% RSLogix 500 project P2.RSS, saved by version 8.30.00.16 %
PROJECT "UNTITLED"    % processor: Bul.1763 MicroLogix 1100 Series B %

PROGRAM FILES
  LAD 2 "MAIN"  3 rungs
  LAD 3 "IO"  9 rungs
  LAD 4 "CONTROLS"  9 rungs

DATA FILES
  O0 OUTPUT  4 elements
  I1 INPUT  6 elements
  S2 STATUS  66 elements
  B3 BINARY  1 elements
  T4 TIMER  2 elements
  C5 COUNTER  1 elements
  R6 CONTROL  1 elements
  N7 INTEGER  1 elements
  F8 FLOAT  1 elements

LADDER 2 "MAIN"
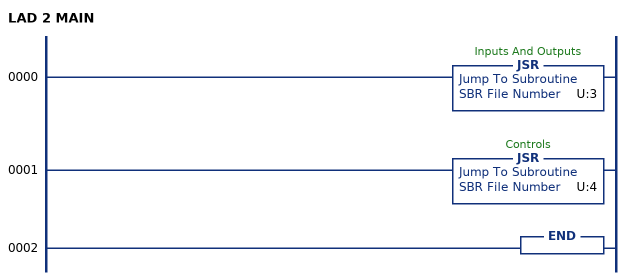
% Rung: 0 %
SOR JSR U:3 EOR
%   U:3  "Inputs And Outputs" %
% Rung: 1 %
SOR JSR U:4 EOR
%   U:4  "Controls" %
% Rung: 2 %
SOR END EOR

LADDER 3 "IO"
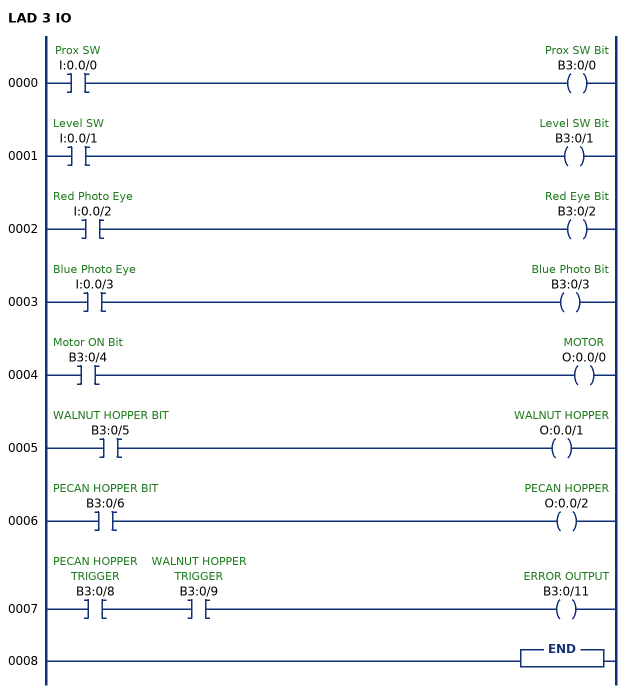
% Rung: 0 %
SOR XIC I:0.0/0 OTE B3:0/0 EOR
%   I:0.0/0  "Prox SW" %
%   B3:0/0  "Prox SW Bit" %
% Rung: 1 %
SOR XIC I:0.0/1 OTE B3:0/1 EOR
%   I:0.0/1  "Level SW" %
%   B3:0/1  "Level SW Bit" %
% Rung: 2 %
SOR XIC I:0.0/2 OTE B3:0/2 EOR
%   I:0.0/2  "Red Photo Eye" %
%   B3:0/2  "Red Eye Bit" %
% Rung: 3 %
SOR XIC I:0.0/3 OTE B3:0/3 EOR
%   I:0.0/3  "Blue Photo Eye" %
%   B3:0/3  "Blue Photo Bit" %
% Rung: 4 %
SOR XIC B3:0/4 OTE O:0.0/0 EOR
%   B3:0/4  "Motor ON Bit" %
%   O:0.0/0  "MOTOR" %
% Rung: 5 %
SOR XIC B3:0/5 OTE O:0.0/1 EOR
%   B3:0/5  "WALNUT HOPPER BIT" %
%   O:0.0/1  "WALNUT HOPPER" %
% Rung: 6 %
SOR XIC B3:0/6 OTE O:0.0/2 EOR
%   B3:0/6  "PECAN HOPPER BIT" %
%   O:0.0/2  "PECAN HOPPER" %
% Rung: 7 %
SOR XIC B3:0/8 XIC B3:0/9 OTE B3:0/11 EOR
%   B3:0/8  "PECAN HOPPER TRIGGER" %
%   B3:0/9  "WALNUT HOPPER TRIGGER" %
%   B3:0/11  "ERROR OUTPUT" %
% Rung: 8 %
SOR END EOR

LADDER 4 "CONTROLS"
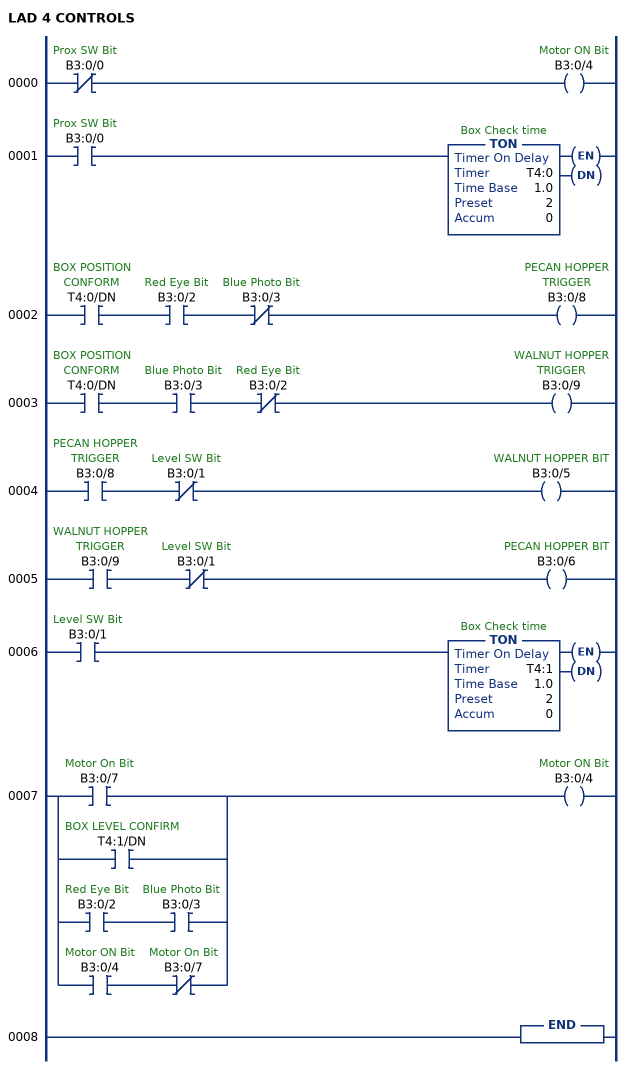
% Rung: 0 %
SOR XIO B3:0/0 OTE B3:0/4 EOR
%   B3:0/0  "Prox SW Bit" %
%   B3:0/4  "Motor ON Bit" %
% Rung: 1 %
SOR XIC B3:0/0 TON T4:0 1.0 2 0 EOR
%   B3:0/0  "Prox SW Bit" %
%   T4:0  "Box Check time" %
% Rung: 2 %
SOR XIC T4:0/DN XIC B3:0/2 XIO B3:0/3 OTE B3:0/8 EOR
%   T4:0/DN  "BOX POSITION CONFORM" %
%   B3:0/2  "Red Eye Bit" %
%   B3:0/3  "Blue Photo Bit" %
%   B3:0/8  "PECAN HOPPER TRIGGER" %
% Rung: 3 %
SOR XIC T4:0/DN XIC B3:0/3 XIO B3:0/2 OTE B3:0/9 EOR
%   T4:0/DN  "BOX POSITION CONFORM" %
%   B3:0/3  "Blue Photo Bit" %
%   B3:0/2  "Red Eye Bit" %
%   B3:0/9  "WALNUT HOPPER TRIGGER" %
% Rung: 4 %
SOR XIC B3:0/8 XIO B3:0/1 OTE B3:0/5 EOR
%   B3:0/8  "PECAN HOPPER TRIGGER" %
%   B3:0/1  "Level SW Bit" %
%   B3:0/5  "WALNUT HOPPER BIT" %
% Rung: 5 %
SOR XIC B3:0/9 XIO B3:0/1 OTE B3:0/6 EOR
%   B3:0/9  "WALNUT HOPPER TRIGGER" %
%   B3:0/1  "Level SW Bit" %
%   B3:0/6  "PECAN HOPPER BIT" %
% Rung: 6 %
SOR XIC B3:0/1 TON T4:1 1.0 2 0 EOR
%   B3:0/1  "Level SW Bit" %
%   T4:1  "Box Check time" %
% Rung: 7 %
SOR BST XIC B3:0/7 NXB BST XIC T4:1/DN NXB BST XIC B3:0/2 XIC B3:0/3 NXB XIC B3:0/4 XIO B3:0/7 BND BND BND OTE B3:0/4 EOR
%   B3:0/7  "Motor On Bit" %
%   T4:1/DN  "BOX LEVEL CONFIRM" %
%   B3:0/2  "Red Eye Bit" %
%   B3:0/3  "Blue Photo Bit" %
%   B3:0/4  "Motor ON Bit" %
% Rung: 8 %
SOR END EOR

OTHER DOCUMENTED ADDRESSES
  B3:0/10  "ERROR BIT"
  N7:0  "Status 1:Belt moving 2:Filling Pecan 3:Filling Walnut 4:Box is filled"
  N7:1  "Status 1:Belt moving 2:Filling Pecan 3:Filling Walnut 4:Box is filled"
  T4:0/0  "Box Check time"
  T4:0/1  "BOX FILL TIME"
  U:5  "Status"

DATA TABLE (non-zero values as saved)
DATA T4
% .PRE .ACC %
% T4:0 % 2 0
% T4:1 % 2 0
